(* CODESYS project 3v12manLoadTestPLC.project

Project tree, tasks and I/O mapping:
  Device : Owen SPK2xx 03.CS.WEB, Owen, order no. 023, version 3.5.4.20
    application Application
      task MainTask (cyclic, interval t#20ms, priority 1) calls PLC_PRG
      task VISU_TASK (cyclic, interval 100 ms, priority 31) calls VisuElems.Visu_Prg
      program PLC_PRG [ST]: actNextUnloadStep, actInit, outWriteVars, autoLoadHopper, autoUnloadHopper, actTimeCounting, sysAutoStat, sysManStat, manLoad, manUnload, inReadVars, setTara, actLoadSwitches, actUnloadSwitches, pause, chkEngines
      image pool ImagePool
      data type TableStruct
      Functions/
        function TimeInput [ST]
        function two_word_to_real [ST]
        function block NoiseFilter [ST]: isInEdges, setEdges, setAccuracy, refresh
      GlobalVarList/
        global variables GVL
        global variables ArrayList
        global variables TimeVars
        global variables CurrentValues
      Windows/
        visualisation Visualization
        visualisation ManualInput
        visualisation Settings
        visualisation AutoWork
        visualisation LoadProcessWindow
        visualisation LoadingFinished
        visualisation UnloadProcessWindow
        visualisation RepeatOrNewPRG
        visualisation TimeCounter
        Dialogs/
          visualisation DialogLoad
          visualisation Alarm
        visualisation TmpUnused
        visualisation SystemSettings
      Managers/
        libraries: VisuDialogs, * (System); CmpSysExec, 1.0.0.2 (Owen); SPK_Tools, 1.0.1 (Owen); RS mode library, 1.0.0.0 (Owen); ArchiverSPK, 3.5.3.53 (Owen); CAA File, 3.5.5.0 (CAA Technical Workgroup); Time and Date, 3.5.1.0 (3S - Smart Software Solutions GmbH); Standard, * (System); Mx110Assistant, 3.5.4.0 (Owen)
        RecipeManager
          recipe definition Receipt: arrayOfIngr[0].stepNum : STRING; arrayOfIngr[0].nameOfIngr : STRING; arrayOfIngr[0].weightOfIngr : STRING; arrayOfIngr[0].isDissolve : STRING; arrayOfIngr[0].timeOfMixing : STRING; arrayOfIngr[0].addMessage : STRING; arrayOfIngr[1].stepNum : STRING; arrayOfIngr[1].nameOfIngr : STRING; arrayOfIngr[1].weightOfIngr : STRING; arrayOfIngr[1].isDissolve : STRING; arrayOfIngr[1].timeOfMixing : STRING; arrayOfIngr[1].addMessage : STRING; arrayOfIngr[2].stepNum : STRING; arrayOfIngr[2].nameOfIngr : STRING; arrayOfIngr[2].weightOfIngr : STRING; arrayOfIngr[2].isDissolve : STRING; arrayOfIngr[2].timeOfMixing : STRING; arrayOfIngr[2].addMessage : STRING; arrayOfIngr[3].stepNum : STRING; arrayOfIngr[3].nameOfIngr : STRING; arrayOfIngr[3].weightOfIngr : STRING; arrayOfIngr[3].isDissolve : STRING; arrayOfIngr[3].timeOfMixing : STRING; arrayOfIngr[3].addMessage : STRING; arrayOfIngr[4].stepNum : STRING; arrayOfIngr[4].nameOfIngr : STRING; arrayOfIngr[4].weightOfIngr : STRING; arrayOfIngr[4].isDissolve : STRING; arrayOfIngr[4].timeOfMixing : STRING; arrayOfIngr[4].addMessage : STRING; arrayOfIngr[5].stepNum : STRING; arrayOfIngr[5].nameOfIngr : STRING; arrayOfIngr[5].weightOfIngr : STRING; arrayOfIngr[5].isDissolve : STRING; arrayOfIngr[5].timeOfMixing : STRING; arrayOfIngr[5].addMessage : STRING; arrayOfIngr[6].stepNum : STRING; arrayOfIngr[6].nameOfIngr : STRING; arrayOfIngr[6].weightOfIngr : STRING; arrayOfIngr[6].isDissolve : STRING; arrayOfIngr[6].timeOfMixing : STRING; arrayOfIngr[6].addMessage : STRING; arrayOfIngr[7].stepNum : STRING; arrayOfIngr[7].nameOfIngr : STRING; arrayOfIngr[7].weightOfIngr : STRING; arrayOfIngr[7].isDissolve : STRING; arrayOfIngr[7].timeOfMixing : STRING; arrayOfIngr[7].addMessage : STRING; arrayOfIngr[8].stepNum : STRING; arrayOfIngr[8].nameOfIngr : STRING; arrayOfIngr[8].weightOfIngr : STRING; arrayOfIngr[8].isDissolve : STRING; arrayOfIngr[8].timeOfMixing : STRING; arrayOfIngr[8].addMessage : STRING; arrayOfIngr[9].stepNum : STRING; arrayOfIngr[9].nameOfIngr : STRING; arrayOfIngr[9].weightOfIngr : STRING; arrayOfIngr[9].isDissolve : STRING; arrayOfIngr[9].timeOfMixing : STRING; arrayOfIngr[9].addMessage : STRING; arrayOfIngr[10].stepNum : STRING; arrayOfIngr[10].nameOfIngr : STRING; arrayOfIngr[10].weightOfIngr : STRING; arrayOfIngr[10].isDissolve : STRING; arrayOfIngr[10].timeOfMixing : STRING; arrayOfIngr[10].addMessage : STRING; arrayOfIngr[11].stepNum : STRING; arrayOfIngr[11].nameOfIngr : STRING; arrayOfIngr[11].weightOfIngr : STRING; arrayOfIngr[11].isDissolve : STRING; arrayOfIngr[11].timeOfMixing : STRING; arrayOfIngr[11].addMessage : STRING; arrayOfIngr[12].stepNum : STRING; arrayOfIngr[12].nameOfIngr : STRING; arrayOfIngr[12].weightOfIngr : STRING; arrayOfIngr[12].isDissolve : STRING; arrayOfIngr[12].timeOfMixing : STRING; arrayOfIngr[12].addMessage : STRING; arrayOfIngr[13].stepNum : STRING; arrayOfIngr[13].nameOfIngr : STRING; arrayOfIngr[13].weightOfIngr : STRING; arrayOfIngr[13].isDissolve : STRING; arrayOfIngr[13].timeOfMixing : STRING; arrayOfIngr[13].addMessage : STRING; arrayOfIngr[14].stepNum : STRING; arrayOfIngr[14].nameOfIngr : STRING; arrayOfIngr[14].weightOfIngr : STRING; arrayOfIngr[14].isDissolve : STRING; arrayOfIngr[14].timeOfMixing : STRING; arrayOfIngr[14].addMessage : STRING; arrayOfIngr[15].stepNum : STRING; arrayOfIngr[15].nameOfIngr : STRING; arrayOfIngr[15].weightOfIngr : STRING; arrayOfIngr[15].isDissolve : STRING; arrayOfIngr[15].timeOfMixing : STRING; arrayOfIngr[15].addMessage : STRING; arrayOfIngr[16].stepNum : STRING; arrayOfIngr[16].nameOfIngr : STRING; arrayOfIngr[16].weightOfIngr : STRING; arrayOfIngr[16].isDissolve : STRING; arrayOfIngr[16].timeOfMixing : STRING; arrayOfIngr[16].addMessage : STRING; arrayOfIngr[17].stepNum : STRING; arrayOfIngr[17].nameOfIngr : STRING; arrayOfIngr[17].weightOfIngr : STRING; arrayOfIngr[17].isDissolve : STRING; arrayOfIngr[17].timeOfMixing : STRING; arrayOfIngr[17].addMessage : STRING; arrayOfIngr[18].stepNum : STRING; arrayOfIngr[18].nameOfIngr : STRING; arrayOfIngr[18].weightOfIngr : STRING; arrayOfIngr[18].isDissolve : STRING; arrayOfIngr[18].timeOfMixing : STRING; arrayOfIngr[18].addMessage : STRING; arrayOfIngr[19].stepNum : STRING; arrayOfIngr[19].nameOfIngr : STRING; arrayOfIngr[19].weightOfIngr : STRING; arrayOfIngr[19].isDissolve : STRING; arrayOfIngr[19].timeOfMixing : STRING; arrayOfIngr[19].addMessage : STRING; arrayOfIngr[20].stepNum : STRING; arrayOfIngr[20].nameOfIngr : STRING; arrayOfIngr[20].weightOfIngr : STRING; arrayOfIngr[20].isDissolve : STRING; arrayOfIngr[20].timeOfMixing : STRING; arrayOfIngr[20].addMessage : STRING; arrayOfIngr[21].stepNum : STRING; arrayOfIngr[21].nameOfIngr : STRING; arrayOfIngr[21].weightOfIngr : STRING; arrayOfIngr[21].isDissolve : STRING; arrayOfIngr[21].timeOfMixing : STRING; arrayOfIngr[21].addMessage : STRING; arrayOfIngr[22].stepNum : STRING; arrayOfIngr[22].nameOfIngr : STRING; arrayOfIngr[22].weightOfIngr : STRING; arrayOfIngr[22].isDissolve : STRING; arrayOfIngr[22].timeOfMixing : STRING; arrayOfIngr[22].addMessage : STRING; arrayOfIngr[23].stepNum : STRING; arrayOfIngr[23].nameOfIngr : STRING; arrayOfIngr[23].weightOfIngr : STRING; arrayOfIngr[23].isDissolve : STRING; arrayOfIngr[23].timeOfMixing : STRING; arrayOfIngr[23].addMessage : STRING; arrayOfIngr[24].stepNum : STRING; arrayOfIngr[24].nameOfIngr : STRING; arrayOfIngr[24].weightOfIngr : STRING; arrayOfIngr[24].isDissolve : STRING; arrayOfIngr[24].timeOfMixing : STRING; arrayOfIngr[24].addMessage : STRING; arrayOfIngr[25].stepNum : STRING; arrayOfIngr[25].nameOfIngr : STRING; arrayOfIngr[25].weightOfIngr : STRING; arrayOfIngr[25].isDissolve : STRING; arrayOfIngr[25].timeOfMixing : STRING; arrayOfIngr[25].addMessage : STRING; arrayOfIngr[26].stepNum : STRING; arrayOfIngr[26].nameOfIngr : STRING; arrayOfIngr[26].weightOfIngr : STRING; arrayOfIngr[26].isDissolve : STRING; arrayOfIngr[26].timeOfMixing : STRING; arrayOfIngr[26].addMessage : STRING; arrayOfIngr[27].stepNum : STRING; arrayOfIngr[27].nameOfIngr : STRING; arrayOfIngr[27].weightOfIngr : STRING; arrayOfIngr[27].isDissolve : STRING; arrayOfIngr[27].timeOfMixing : STRING; arrayOfIngr[27].addMessage : STRING; arrayOfIngr[28].stepNum : STRING; arrayOfIngr[28].nameOfIngr : STRING; arrayOfIngr[28].weightOfIngr : STRING; arrayOfIngr[28].isDissolve : STRING; arrayOfIngr[28].timeOfMixing : STRING; arrayOfIngr[28].addMessage : STRING; arrayOfIngr[29].stepNum : STRING; arrayOfIngr[29].nameOfIngr : STRING; arrayOfIngr[29].weightOfIngr : STRING; arrayOfIngr[29].isDissolve : STRING; arrayOfIngr[29].timeOfMixing : STRING; arrayOfIngr[29].addMessage : STRING; arrayOfIngr[30].stepNum : STRING; arrayOfIngr[30].nameOfIngr : STRING; arrayOfIngr[30].weightOfIngr : STRING; arrayOfIngr[30].isDissolve : STRING; arrayOfIngr[30].timeOfMixing : STRING; arrayOfIngr[30].addMessage : STRING; arrayOfIngr[31].stepNum : STRING; arrayOfIngr[31].nameOfIngr : STRING; arrayOfIngr[31].weightOfIngr : STRING; arrayOfIngr[31].isDissolve : STRING; arrayOfIngr[31].timeOfMixing : STRING; arrayOfIngr[31].addMessage : STRING; arrayOfIngr[32].stepNum : STRING; arrayOfIngr[32].nameOfIngr : STRING; arrayOfIngr[32].weightOfIngr : STRING; arrayOfIngr[32].isDissolve : STRING; arrayOfIngr[32].timeOfMixing : STRING; arrayOfIngr[32].addMessage : STRING; arrayOfIngr[33].stepNum : STRING; arrayOfIngr[33].nameOfIngr : STRING; arrayOfIngr[33].weightOfIngr : STRING; arrayOfIngr[33].isDissolve : STRING; arrayOfIngr[33].timeOfMixing : STRING; arrayOfIngr[33].addMessage : STRING; arrayOfIngr[34].stepNum : STRING; arrayOfIngr[34].nameOfIngr : STRING; arrayOfIngr[34].weightOfIngr : STRING; arrayOfIngr[34].isDissolve : STRING; arrayOfIngr[34].timeOfMixing : STRING; arrayOfIngr[34].addMessage : STRING; arrayOfIngr[35].stepNum : STRING; arrayOfIngr[35].nameOfIngr : STRING; arrayOfIngr[35].weightOfIngr : STRING; arrayOfIngr[35].isDissolve : STRING; arrayOfIngr[35].timeOfMixing : STRING; arrayOfIngr[35].addMessage : STRING; arrayOfIngr[36].stepNum : STRING; arrayOfIngr[36].nameOfIngr : STRING; arrayOfIngr[36].weightOfIngr : STRING; arrayOfIngr[36].isDissolve : STRING; arrayOfIngr[36].timeOfMixing : STRING; arrayOfIngr[36].addMessage : STRING; arrayOfIngr[37].stepNum : STRING; arrayOfIngr[37].nameOfIngr : STRING; arrayOfIngr[37].weightOfIngr : STRING; arrayOfIngr[37].isDissolve : STRING; arrayOfIngr[37].timeOfMixing : STRING; arrayOfIngr[37].addMessage : STRING; arrayOfIngr[38].stepNum : STRING; arrayOfIngr[38].nameOfIngr : STRING; arrayOfIngr[38].weightOfIngr : STRING; arrayOfIngr[38].isDissolve : STRING; arrayOfIngr[38].timeOfMixing : STRING; arrayOfIngr[38].addMessage : STRING; arrayOfIngr[39].stepNum : STRING; arrayOfIngr[39].nameOfIngr : STRING; arrayOfIngr[39].weightOfIngr : STRING; arrayOfIngr[39].isDissolve : STRING; arrayOfIngr[39].timeOfMixing : STRING; arrayOfIngr[39].addMessage : STRING; arrayOfIngr[40].stepNum : STRING; arrayOfIngr[40].nameOfIngr : STRING; arrayOfIngr[40].weightOfIngr : STRING; arrayOfIngr[40].isDissolve : STRING; arrayOfIngr[40].timeOfMixing : STRING; arrayOfIngr[40].addMessage : STRING; arrayOfIngr[41].stepNum : STRING; arrayOfIngr[41].nameOfIngr : STRING; arrayOfIngr[41].weightOfIngr : STRING; arrayOfIngr[41].isDissolve : STRING; arrayOfIngr[41].timeOfMixing : STRING; arrayOfIngr[41].addMessage : STRING; arrayOfIngr[42].stepNum : STRING; arrayOfIngr[42].nameOfIngr : STRING; arrayOfIngr[42].weightOfIngr : STRING; arrayOfIngr[42].isDissolve : STRING; arrayOfIngr[42].timeOfMixing : STRING; arrayOfIngr[42].addMessage : STRING; arrayOfIngr[43].stepNum : STRING; arrayOfIngr[43].nameOfIngr : STRING; arrayOfIngr[43].weightOfIngr : STRING; arrayOfIngr[43].isDissolve : STRING; arrayOfIngr[43].timeOfMixing : STRING; arrayOfIngr[43].addMessage : STRING; arrayOfIngr[44].stepNum : STRING; arrayOfIngr[44].nameOfIngr : STRING; arrayOfIngr[44].weightOfIngr : STRING; arrayOfIngr[44].isDissolve : STRING; arrayOfIngr[44].timeOfMixing : STRING; arrayOfIngr[44].addMessage : STRING; arrayOfIngr[45].stepNum : STRING; arrayOfIngr[45].nameOfIngr : STRING; arrayOfIngr[45].weightOfIngr : STRING; arrayOfIngr[45].isDissolve : STRING; arrayOfIngr[45].timeOfMixing : STRING; arrayOfIngr[45].addMessage : STRING; arrayOfIngr[46].stepNum : STRING; arrayOfIngr[46].nameOfIngr : STRING; arrayOfIngr[46].weightOfIngr : STRING; arrayOfIngr[46].isDissolve : STRING; arrayOfIngr[46].timeOfMixing : STRING; arrayOfIngr[46].addMessage : STRING; arrayOfIngr[47].stepNum : STRING; arrayOfIngr[47].nameOfIngr : STRING; arrayOfIngr[47].weightOfIngr : STRING; arrayOfIngr[47].isDissolve : STRING; arrayOfIngr[47].timeOfMixing : STRING; arrayOfIngr[47].addMessage : STRING; arrayOfIngr[48].stepNum : STRING; arrayOfIngr[48].nameOfIngr : STRING; arrayOfIngr[48].weightOfIngr : STRING; arrayOfIngr[48].isDissolve : STRING; arrayOfIngr[48].timeOfMixing : STRING; arrayOfIngr[48].addMessage : STRING; arrayOfIngr[49].stepNum : STRING; arrayOfIngr[49].nameOfIngr : STRING; arrayOfIngr[49].weightOfIngr : STRING; arrayOfIngr[49].isDissolve : STRING; arrayOfIngr[49].timeOfMixing : STRING; arrayOfIngr[49].addMessage : STRING; arrayOfIngr[50].stepNum : STRING; arrayOfIngr[50].nameOfIngr : STRING; arrayOfIngr[50].weightOfIngr : STRING; arrayOfIngr[50].isDissolve : STRING; arrayOfIngr[50].timeOfMixing : STRING; arrayOfIngr[50].addMessage : STRING
      Classes/
        function block List [ST]: getPrgIdx, getLineFromPrgArr, checkPrgArr, clearList, clearLine, writeLine
        function block DiscrSwitch [ST]: allOff, set, setLaterOn, setLaterOff, unloadOn, unloadLaterOff, unloadOff
        function block Checker [ST]: isHopperEmpty, isPrgActive
        function block Way [ST]: getWay, tmpLimitWay, getWayId, setWay, setIdx
    COM_2 : Modbus COM, 3S - Smart Software Solutions GmbH, version 3.4.0.0
        settings: DataBits = 8; StopBits = 1; ComPort = 3
      Modbus_Master_COM_Port_2 : Modbus Master, COM Port, 3S - Smart Software Solutions GmbH, version 3.5.5.0
          settings: Transmission = 'RTU'; ResponseTimeout = 300; TimeBetweenFrames = 20; Auto-restart communication = TRUE
        Out_MU110_16R : Modbus Slave, COM Port, 3S - Smart Software Solutions GmbH, version 3.5.4.0
            settings: SlaveAddress = 17; ResponseTimeout = 300; UseExtendedFunctionCodes = TRUE; Channel 0.Function Code = 16; Channel 0.Read Offset = 0; Channel 0.Read Length = 0; Channel 0.Write Offset = 16#0032; Channel 0.Write Length = 1; Channel 0.Cycle Time = 100
            output Application.iOutDiscrets : ARRAY[0..0] OF WORD  // Channel 0
        In_MV110_16D : Modbus Slave, COM Port, 3S - Smart Software Solutions GmbH, version 3.5.4.0
            settings: SlaveAddress = 1; ResponseTimeout = 300; UseExtendedFunctionCodes = TRUE; Channel 0.Function Code = 3; Channel 0.Read Offset = 16#0033; Channel 0.Read Length = 1; Channel 0.Write Offset = 0; Channel 0.Write Length = 0; Channel 0.Cycle Time = 100
            input  Application.iInDiscrets : ARRAY[0..0] OF WORD  // Channel 0
    COM_3 : Modbus COM, 3S - Smart Software Solutions GmbH, version 3.4.0.0
        settings: DataBits = 8; StopBits = 1; ComPort = 4
      Modbus_Master_COM_Port : Modbus Master, COM Port, 3S - Smart Software Solutions GmbH, version 3.5.5.0
          settings: Transmission = 'RTU'; ResponseTimeout = 300; TimeBetweenFrames = 10; Auto-restart communication = TRUE
        MV110_1TD : MV110-1TD, Owen, order no. 3.5.4.1, version 3.5.4.0
            settings: SlaveAddress = 1; ResponseTimeout = 300; UseExtendedFunctionCodes = TRUE
            unmapped channels: Rd.fF1, Rd.St, in1, out1
  text list GlobalTextList
  GlobalImagePool
  image pool ImagePool
  5ce3da45-db07-42e7-a21c-a00fff4ed8f6|C:\Users\Валентин\Desktop\home.png
  5ce3da45-db07-42e7-a21c-a00fff4ed8f6|D:\Pictures\tanzania.jpg
  5ce3da45-db07-42e7-a21c-a00fff4ed8f6|D:\Pictures\tanzania800x480.jpg
  5ce3da45-db07-42e7-a21c-a00fff4ed8f6|D:\Pictures\BeachHouse800x480.jpg
  5ce3da45-db07-42e7-a21c-a00fff4ed8f6|D:\Projects\OWEN\JAVA\GIT\settings.png
  5ce3da45-db07-42e7-a21c-a00fff4ed8f6|D:\Projects\OWEN\PIC\motherboard.png
  5ce3da45-db07-42e7-a21c-a00fff4ed8f6|D:\Projects\OWEN\PIC\home.png
  5ce3da45-db07-42e7-a21c-a00fff4ed8f6|D:\Projects\OWEN\PIC\settings.jpg
  5ce3da45-db07-42e7-a21c-a00fff4ed8f6|D:\Projects\OWEN\PIC\reset.jpg
  5ce3da45-db07-42e7-a21c-a00fff4ed8f6|D:\Projects\OWEN\PIC\reset.png
  5ce3da45-db07-42e7-a21c-a00fff4ed8f6|D:\Projects\OWEN\PIC\resetButton.png
  5ce3da45-db07-42e7-a21c-a00fff4ed8f6|D:\Projects\OWEN\PIC\start.png
  5ce3da45-db07-42e7-a21c-a00fff4ed8f6|D:\Projects\OWEN\PIC\remove.png
  5ce3da45-db07-42e7-a21c-a00fff4ed8f6|D:\Projects\OWEN\PIC\ok.png
  5ce3da45-db07-42e7-a21c-a00fff4ed8f6|D:\Projects\OWEN\PIC\cancel.png
  function block Time_Struct [ST]
  5ce3da45-db07-42e7-a21c-a00fff4ed8f6|D:\Projects\OWEN\PIC\add.png
  5ce3da45-db07-42e7-a21c-a00fff4ed8f6|D:\Projects\OWEN\PIC\back.png
  5ce3da45-db07-42e7-a21c-a00fff4ed8f6|D:\Projects\OWEN\PIC\next.png
  5ce3da45-db07-42e7-a21c-a00fff4ed8f6|D:\Projects\OWEN\PIC\Drives-Downloads-icon.png
  5ce3da45-db07-42e7-a21c-a00fff4ed8f6|D:\Projects\OWEN\PIC\Actions-application-exit-icon.png
  5ce3da45-db07-42e7-a21c-a00fff4ed8f6|D:\Projects\OWEN\PIC\App-desktop-enhancements-icon.png
  5ce3da45-db07-42e7-a21c-a00fff4ed8f6|D:\Projects\OWEN\PIC\chemistryS.png
  5ce3da45-db07-42e7-a21c-a00fff4ed8f6|D:\Projects\OWEN\PIC\chemistry.png
  5ce3da45-db07-42e7-a21c-a00fff4ed8f6|D:\Projects\OWEN\PIC\Iconshock-Real-Vista-Education-Laboratory.png
  5ce3da45-db07-42e7-a21c-a00fff4ed8f6|D:\Projects\OWEN\PIC\pause.png
  5ce3da45-db07-42e7-a21c-a00fff4ed8f6|D:\Projects\OWEN\PIC\startAgain.png
  5ce3da45-db07-42e7-a21c-a00fff4ed8f6|D:\Projects\OWEN\PIC\start-button-305427_960_720.png
  5ce3da45-db07-42e7-a21c-a00fff4ed8f6|D:\Projects\OWEN\PIC\repeat.png
  5ce3da45-db07-42e7-a21c-a00fff4ed8f6|D:\Projects\OWEN\PIC\download.png
  5ce3da45-db07-42e7-a21c-a00fff4ed8f6|D:\Projects\OWEN\PIC\upload.png
*)

// Device/Application/TableStruct
TYPE TableStruct :
STRUCT
	stepNum:STRING;
	nameOfIngr:STRING;
	weightOfIngr:STRING;
	isDissolve:STRING;
	timeOfMixing:STRING;
	addMessage:STRING;	
END_STRUCT
END_TYPE

// Device/Application/GlobalVarList/GVL
VAR_GLOBAL
	iOutDiscrets: INT;
	iInDiscrets:INT;
	ON : BOOL := TRUE;
	OFF : BOOL := FALSE;	
	arr1:ARRAY[0..1]OF WORD;		
	arr2:ARRAY[0..1]OF WORD;
	arr3:ARRAY[0..1]OF WORD;
	arr4:ARRAY[0..1]OF WORD;	
END_VAR

// Device/Application/GlobalVarList/ArrayList
VAR_GLOBAL
	ListOfPrgNames: ARRAY[0..100] OF STRING;	
	ptToListPrg: POINTER TO ARRAY [0..100] OF STRING := ADR(ListOfPrgNames);
	arrayOfIngr: ARRAY[0..50] OF TableStruct;
	tempArrOfIngr: ARRAY[0..100] OF TableStruct;		
END_VAR

// Device/Application/GlobalVarList/TimeVars
VAR_GLOBAL
	timerActive:BOOL := FALSE;
	strTimer:STRING;
	inputTime:DWORD;
END_VAR

// Device/Application/GlobalVarList/CurrentValues
VAR_GLOBAL
	currentPrgSteps:INT;	
	currentProgramIdx:INT;
	currentPrgName: STRING;
	currentIngredientName: STRING;
	currentWeight: INT;
	currentPoint : INT;
//	strCrntWay: STRING;
	message: STRING;	
	currentTimeMixing: TIME;
END_VAR

// Device/Application/PLC_PRG
PROGRAM PLC_PRG
VAR
	iMaxWeight: INT := 1000;	

	tOn1:TON;
	tOn2:TON;
	tCheckDelay:TON;
	
	switch:DiscrSwitch;
	ptSwitch: POINTER TO DiscrSwitch := ADR(switch);
	timeStruct:Time_Struct;	
	bTimerActive:BOOL := FALSE;
	strTimer:STRING;
	dwInTime:DWORD;
	rWeight:REAL;
	
	list:List;
	checker:Checker;
	signalFilter:NoiseFilter;

	strResipesExt:STRING := 'Receipt';
	RecManager:RecipeManCommands;

	bInit:BOOL := TRUE;
	bPause:BOOL;
	bRunOnce:BOOL;
	bLoadDone:BOOL;
	bManLoadDone:BOOL;
	bMsgVisible:BOOL := TRUE;
	bManMode: BOOL;
	
	iTotalIngrWeight:INT;
	iErrEngineNum:INT := 0;
	
	x: INT := 0;
	iEdge: INT := 1000;
	bSwitch: BOOL;
	bLamp: BOOL;	

	data0:REAL;
END_VAR
VAR RETAIN
	rTara:REAL;	
END_VAR

inReadVars();

IF bInit THEN // run once
	actInit();END_IF


IF bManMode THEN
	sysManStat();
ELSE
	sysAutoStat();
END_IF
outWriteVars();

chkEngines();
//data0:=two_word_to_real(ADR(arr1));

ACTION actNextUnloadStep:
bTimerActive := FALSE;
VisuElems.CURRENTVISU := 'UnloadProcessWindow';
currentProgramIdx := currentProgramIdx + 1;
list.getLineFromPrgArr(currentProgramIdx);
IF currentPrgSteps >= currentProgramIdx THEN
		 VisuElems.CURRENTVISU := 'RepeatOrNewPRG';
		 bLoadDone := FALSE;
END_IF
END_ACTION

ACTION actInit:
RecManager.ReloadRecipes(strResipesExt);
RecManager.GetRecipeNames(strResipesExt, ptToListPrg, 100,0);
list(ptToSwitch := ptSwitch);
bInit := FALSE;
END_ACTION

ACTION outWriteVars:

iOutDiscrets := Switch.iOut;
END_ACTION

ACTION autoLoadHopper:
IF bSwitch THEN
  IF x < currentPoint + currentWeight AND x < iMaxWeight THEN 
	 bMsgVisible := FALSE;
	 switch.set(ON);
	 pause();
//	 x := x + 1;	 
  ELSE 
	switch.set(OFF);
	actLoadSwitches();
	IF tOn2.Q THEN
 		currentPoint := currentPoint + currentWeight;
 		IF x >= currentPoint AND currentPrgSteps - 1 > currentProgramIdx THEN
	 		currentProgramIdx := currentProgramIdx + 1;
	 		list.getLineFromPrgArr(currentProgramIdx);
		 ELSIF currentPrgSteps >= currentProgramIdx THEN
		 	currentProgramIdx := 0;
		 	list.getLineFromPrgArr(currentProgramIdx);
		 	bLoadDone:=TRUE;
		 	VisuElems.CURRENTVISU := 'LoadingFinished';
		END_IF
 		bMsgVisible := TRUE;
		bSwitch := FALSE;		
	END_IF
 END_IF
END_IF
END_ACTION

ACTION autoUnloadHopper:
IF bSwitch THEN
  IF x > currentPoint - currentWeight AND x > 0 THEN 
	 bMsgVisible := FALSE;
//	 x := x - 1;
	 Switch.unloadOn();
  ELSE
	actUnloadSwitches();
	IF tOn1.Q THEN	 
 	currentPoint:= currentPoint - currentWeight;
 		IF x >= currentPoint AND currentPrgSteps - 1 >= currentProgramIdx THEN
			VisuElems.CURRENTVISU := 'TimeCounter';
			bTimerActive:=TRUE;	  
		END_IF
 	bMsgVisible := TRUE;
 	bSwitch:= FALSE;
	tOn1(IN := FALSE);
	END_IF	
 END_IF
END_IF
END_ACTION

ACTION actTimeCounting:
IF TIME_TO_REAL(currentTimeMixing) >= 0 THEN
 	currentTimeMixing := REAL_TO_TIME ( TIME_TO_REAL(currentTimeMixing) - 20); 
	timeStruct(Type_Time := currentTimeMixing);
	strTimer:=CONCAT(CONCAT(DWORD_TO_STRING(timeStruct.Minute),'m:'),CONCAT(DWORD_TO_STRING(timeStruct.Second),'s'));
		IF TIME_TO_REAL(currentTimeMixing) = 0 THEN
			actNextUnloadStep();
		END_IF	
END_IF
END_ACTION

ACTION sysAutoStat:
IF bTimerActive THEN 
	actTimeCounting(); 
END_IF

IF bLoadDone THEN	
	autoUnloadHopper();
ELSE	
	autoLoadHopper();
END_IF
END_ACTION

ACTION sysManStat:
IF bManLoadDone THEN	
	manUnload();
ELSE
	manLoad();
END_IF
END_ACTION

ACTION manLoad:
IF bRunOnce THEN
		tOn1(IN := FALSE);
		list.way.getWay();
		switch(iWayIdx := list.way.getWayId());
		bRunOnce := FALSE;
END_IF
IF bSwitch THEN	
  IF x < currentWeight AND x < iMaxWeight THEN 
	Switch.set(ON);	
//	x := x + 1;	 
  ELSE
	switch.set(OFF);
//actLoadSwitches();
 END_IF
END_IF
END_ACTION

ACTION manUnload:
IF bSwitch THEN
  IF x > 0 THEN 
	 switch.unloadOn();
//	 x := x - 1;	 
  ELSE
	  
	//switch.unloadOff();
	actUnloadSwitches();
	tOn1(IN := bSwitch);
 END_IF
END_IF
END_ACTION

ACTION inReadVars:
rWeight := MV110_1TD.RdfF1 - rTara;
signalFilter(rIn := rWeight, rOut => rWeight);
x := REAL_TO_INT(rWeight);
//IF iInDiscrets.0 THEN
	//bSwitch := TRUE;
//END_IF
switch(iIn := iInDiscrets);
END_ACTION

ACTION setTara:
rTara := MV110_1TD.RdfF1;
signalFilter.refresh();
END_ACTION

ACTION actLoadSwitches:
switch.set(OFF);
tOn1(IN := TRUE, PT := T#1S);
switch.setLaterOn(tOn1.Q);
tOn2(IN := tOn1.Q, PT := T#10S);
	IF tOn2.Q THEN
		switch.setLaterOff(OFF);
		bSwitch := FALSE;
		tOn1(IN := FALSE);
	END_IF
END_ACTION

ACTION actUnloadSwitches:
switch.set(OFF);
switch.unloadOff();
tOn1(IN := TRUE, PT := T#10S);	  	  
 	IF tOn1.Q THEN
	 Switch.unloadLaterOff(OFF);
	 bSwitch := FALSE;
	END_IF
END_ACTION

ACTION pause:
IF bPause THEN
	switch.allOff();
END_IF
END_ACTION

ACTION chkEngines:
// проверка подключения автоматов защиты двигателей
tCheckDelay(PT := T#10s, IN := TRUE);
IF tCheckDelay.Q THEN
	IF NOT switch.iIn.12 THEN
		switch.allOff();
		iErrEngineNum := 13;
		VisuElems.CURRENTVISU := 'Alarm';	
	END_IF
	IF NOT switch.iIn.13 THEN	
		switch.allOff();
		iErrEngineNum := 14;
		VisuElems.CURRENTVISU := 'Alarm';	
	END_IF
	IF NOT switch.iIn.14 THEN	
		switch.allOff();
		iErrEngineNum := 15;
		VisuElems.CURRENTVISU := 'Alarm';	
	END_IF
	IF NOT switch.iIn.15 THEN	
		switch.allOff();
		iErrEngineNum := 16;
		VisuElems.CURRENTVISU := 'Alarm';	
	END_IF
END_IF
END_ACTION

END_PROGRAM

// Device/Application/Functions/two_word_to_real
FUNCTION two_word_to_real : REAL
VAR_INPUT
	in_data: POINTER TO ARRAY[0..1]OF WORD;
END_VAR
VAR
	p1:POINTER TO BYTE;
	p2:POINTER TO BYTE;
END_VAR

p1:=ADR(two_word_to_real);
p2:=ADR(in_data^[1]);

p1^:=p2^;
p1:=p1+1;
p2:=p2+1;
p1^:=p2^;
p1:=p1+1;
p2:=ADR(in_data^[0]);
p1^:=p2^;
p1:=p1+1;
p2:=p2+1;
p1^:=p2^;

END_FUNCTION

// Device/Application/Classes/DiscrSwitch

FUNCTION_BLOCK PUBLIC DiscrSwitch
VAR_INPUT
	iIn:INT;	
	iWayIdx:INT;
END_VAR
VAR_OUTPUT
	iOut:INT;
END_VAR

//выключает все 16 переключателей
METHOD allOff
VAR_INPUT
END_VAR
iOut := 0;
END_METHOD

//устанавливает выключатели в ON немедленно
METHOD PUBLIC set
VAR_INPUT
	bInput:BOOL;
END_VAR
CASE iWayIdx OF //набор переключателей в зависимости от текущего пути
	0:// путь по умолчанию		
			iOut.12 := bInput; // двигатель
			iOut.0 := bInput;  //задвижка
			
	1:// путь через вибросито
			iOut.0 := bInput; // двигатель
			iOut.1 := bInput; // двигатель
			iOut.9 := bInput;  //задвижка
			
	2..10://через BigBag
	;
	
END_CASE
END_METHOD

//устанавливает выключатели в ON через интервал
METHOD PUBLIC setLaterOn
VAR_INPUT
	bInput:BOOL;
END_VAR
VAR
END_VAR
CASE iWayIdx OF //набор переключателей в зависимости от текущего пути
	0:// путь по умолчанию
			iOut.3 := bInput; // двигатель					
			iOut.7 := bInput; //распределитель
			iOut.11 := bInput;  //задвижка	
	1:// путь через вибросито
//			iOut.0 := bInput;//двигатель	
			iOut.1 := bInput;  //двигатель
			iOut.6 := bInput; //распределитель
			iOut.9 := bInput;  //задвижка	
	2..10:
	;
	
	ELSE
		;//выброс ошибки на недопустимый параметр	
END_CASE
END_METHOD

//устанавливает выключатели в OFF через интервал
METHOD PUBLIC setLaterOff
VAR_INPUT
	bInput:BOOL;
END_VAR
CASE iWayIdx OF //набор переключателей в зависимости от текущего пути
	0:// путь по умолчанию
			iOut.3 := bInput; // двигатель					
			iOut.7 := bInput; //распределитель
			iOut.11 := bInput;  //задвижка	
	1:// путь через вибросито
//			iOut.0 := bInput;//двигатель	
			iOut.1 := bInput;  //двигатель
			iOut.6 := bInput; //распределитель
			iOut.9 := bInput;  //задвижка
	2..10:
	;
	
	ELSE
		;//выброс ошибки на недопустимый параметр	
END_CASE
END_METHOD

METHOD PUBLIC unloadOn
VAR_INPUT
END_VAR
iOut.1 := TRUE;
iOut.15 := TRUE;
END_METHOD

METHOD unloadLaterOff
VAR_INPUT
	bInput:BOOL;
END_VAR
iOut.15 := bInput;
END_METHOD

METHOD PUBLIC unloadOff
VAR_INPUT
END_VAR
iOut.1 := FALSE;
END_METHOD

END_FUNCTION_BLOCK

// Time_Struct
FUNCTION_BLOCK Time_Struct
VAR_INPUT
	Type_Time:TIME;
END_VAR
VAR_OUTPUT
	Day:DWORD;
	Hour:DWORD;
	Minute:DWORD;
	Second:DWORD;
	Millisecond:DWORD;  
END_VAR
VAR
		Time_DWORD:DWORD;
		Day_Ost:DWORD;
		Hour_Ost:DWORD;
		Minute_Ost:DWORD;
		Second_Ost:DWORD;
		Millisecond_Ost:DWORD; 
END_VAR


Time_DWORD := TIME_TO_DWORD(Type_Time);

Millisecond := Second_Ost;

Second := Minute_Ost/ 1000;
Second_Ost := Minute_Ost MOD 1000;

Minute := Hour_Ost/60000;
Minute_Ost := Hour_Ost MOD 60000;

Hour := Day_Ost/3600000;
Hour_Ost := Day_Ost MOD 3600000;

Day := Time_DWORD/86400000;
Day_Ost := Time_DWORD MOD 86400000;

END_FUNCTION_BLOCK

// Device/Application/Classes/List
FUNCTION_BLOCK List
VAR_INPUT
	ptToSwitch:POINTER TO DiscrSwitch;		
END_VAR
VAR_OUTPUT
END_VAR
VAR	
	way:Way;
	iLinePrgList:INT;
	iLine:INT;	
	iArrLength: INT := 50;
	iPrgAmount:INT := 100;	
	iTotalWeight:INT;
	iCleanIdx:INT;
END_VAR

METHOD getPrgIdx : INT
VAR_INPUT
END_VAR
getPrgIdx := iLinePrgList;
END_METHOD

METHOD PUBLIC getLineFromPrgArr : BOOL
VAR_INPUT
	i:INT;
END_VAR
currentIngredientName := arrayOfIngr[i].nameOfIngr;
currentWeight := STRING_TO_INT(arrayOfIngr[i].weightOfIngr);
//strCrntWay := arrayOfIngr[i].isDissolve;
way.setWay(arrayOfIngr[i].isDissolve);
ptToSwitch^.iWayIdx := way.getWayId();
currentTimeMixing := STRING_TO_TIME(arrayOfIngr[i].timeOfMixing);
message := arrayOfIngr[i].addMessage;
END_METHOD

METHOD PUBLIC checkPrgArr : BOOL
VAR_INPUT
END_VAR
currentProgramIdx:=0;
currentPrgSteps := 0;
iTotalWeight := 0;
IF LEN(arrayOfIngr[0].stepNum) = 0 THEN
		(* Поставить выброс ошибки в ответ на пустую или неправильную программу*)
		RETURN;		
END_IF
	
FOR iLine:=0 TO 100 DO		
	IF 	LEN(arrayOfIngr[iLine].stepNum) > 0 THEN
		currentPrgSteps := currentPrgSteps + 1;
		iTotalWeight := iTotalWeight + STRING_TO_INT(arrayOfIngr[iLine].weightOfIngr);
		(* Поставить выброс ошибки если вес превышает максимально допустимый *)
	ELSE
		RETURN;	
	END_IF
END_FOR
END_METHOD

METHOD PUBLIC clearList : BOOL
VAR_INPUT
END_VAR
FOR iCleanIdx:=0 TO iArrLength DO
	arrayOfIngr[iCleanIdx].stepNum:='';
	arrayOfIngr[iCleanIdx].nameOfIngr:='';
	arrayOfIngr[iCleanIdx].weightOfIngr:='';
	arrayOfIngr[iCleanIdx].isDissolve:='';
	arrayOfIngr[iCleanIdx].timeOfMixing:='';
	arrayOfIngr[iCleanIdx].addMessage:='';
END_FOR
 iCleanIdx:=0;
 iLine:=0;
END_METHOD

METHOD PUBLIC clearLine : BOOL
VAR_INPUT
END_VAR
IF iLine > 0 THEN
	iLine:=iLine - 1;
END_IF
arrayOfIngr[iLine].stepNum:='';
arrayOfIngr[iLine].nameOfIngr:='';
arrayOfIngr[iLine].weightOfIngr:='';
arrayOfIngr[iLine].isDissolve:='';
arrayOfIngr[iLine].timeOfMixing:='';
arrayOfIngr[iLine].addMessage:='';
END_METHOD

METHOD PUBLIC writeLine : BOOL
VAR_INPUT
END_VAR
arrayOfIngr[iLine].stepNum := CONCAT('Step ', INT_TO_STRING(iLine+1));
arrayOfIngr[iLine].nameOfIngr := currentIngredientName;
arrayOfIngr[iLine].weightOfIngr := INT_TO_STRING(currentWeight);
arrayOfIngr[iLine].isDissolve := way.getWay();
currentTimeMixing := TimeInput(inputTime);
arrayOfIngr[iLine].timeOfMixing := TIME_TO_STRING(currentTimeMixing);
arrayOfIngr[iLine].addMessage := message;

iLine := iLine + 1;	
IF iLine > iArrLength THEN
	iLine := 0;
END_IF
END_METHOD

END_FUNCTION_BLOCK

// Device/Application/Classes/Way
//Блок для работы с различными путями поступления ингредиентов в хоппер
FUNCTION_BLOCK Way
VAR_INPUT
END_VAR
VAR_OUTPUT
END_VAR
VAR
	iIdx:INT;
	wayList:ARRAY[0..10] OF STRING := ['Simple', 'Vibro', 'BigBag1', 'BigBag2', 'BigBag3', 'BigBag4','','','','',''];	
END_VAR

//возвращает имя текущего пути
METHOD getWay : STRING
VAR_INPUT
END_VAR
tmpLimitWay();
getWay := wayList[iIdx];
END_METHOD

METHOD PRIVATE tmpLimitWay : BOOL
VAR_INPUT
END_VAR
IF iIdx > 1 THEN
	iIdx := 1;
END_IF
END_METHOD

//Возвращает индекс текущего пути
METHOD PUBLIC getWayId : INT
VAR_INPUT
END_VAR
VAR
END_VAR
tmpLimitWay();
getWayId := iIdx;
END_METHOD

//устанавливает текущий активный путь
METHOD PUBLIC setWay : INT
VAR_INPUT
	strWay:STRING;
END_VAR
VAR
	i:INT;
END_VAR
IF LEN(strWay) = 0 THEN
	iIdx := 0;
	RETURN;
END_IF 
FOR i := 0 TO 10 DO
	IF strWay = wayList[i] THEN  //если нашли соответственное слово в массиве, устанавливаем текущий индекс этого слова
		setIdx(i);
		tmpLimitWay();
		RETURN;
	END_IF
END_FOR
END_METHOD

METHOD PRIVATE setIdx : BOOL
VAR_INPUT
	iIn:INT;
END_VAR
tmpLimitWay();
iIdx := iIn;
END_METHOD

END_FUNCTION_BLOCK

// Device/Application/Functions/TimeInput
//конвертирует DWORD во время в секундах
FUNCTION TimeInput : TIME
VAR_INPUT
	timeSet:DWORD;	
END_VAR
VAR		
END_VAR

TimeInput := DWORD_TO_TIME(timeSet * 1000);

END_FUNCTION

// Device/Application/Classes/Checker
//Проверка условий в программе
FUNCTION_BLOCK Checker
VAR_INPUT	
END_VAR
VAR_OUTPUT	
END_VAR
VAR
END_VAR

//индикатор наличия продукта в хоппере
METHOD isHopperEmpty : BOOL
VAR_INPUT
	iWeightInHopper:INT;
END_VAR
IF iWeightInHopper > 0 THEN
	isHopperEmpty := FALSE;
	ELSE
	isHopperEmpty := TRUE;
END_IF
END_METHOD

//индикатор выбранной программы
METHOD isPrgActive : BOOL
VAR_INPUT
END_VAR
IF LEN(arrayOfIngr[0].stepNum) = 0 THEN
	isPrgActive := FALSE;
	ELSE
	isPrgActive := TRUE;
END_IF
END_METHOD

END_FUNCTION_BLOCK

// Device/Application/Functions/NoiseFilter
//устраняет шумовые колебания сигнала
FUNCTION_BLOCK PUBLIC NoiseFilter
VAR_INPUT
	rIn:REAL;
	tmrStab:TON;
END_VAR
VAR_OUTPUT
	rOut:REAL;
END_VAR
VAR	
	uiMeasureAttempts: UINT := 50;
	rBig:REAL := 1;
	rSmall:REAL := 0.2;
	uiStabCount: UINT := 0;
	rUp:REAL ;
	rLow:REAL;
	bFluct:BOOL;
END_VAR

IF (isInEdges()) THEN
	IF (bFluct) THEN
		RETURN;
	ELSE		
		rOut := rIn;
		uiStabCount := uiStabCount + 1;
		IF uiStabCount > uiMeasureAttempts AND isInEdges()  THEN	
			setEdges(rBig);	
			bFluct := TRUE;
			RETURN;
		END_IF
		setEdges(rSmall);
	END_IF
ELSE
	uiStabCount := 0;
	bFluct := FALSE;
	setEdges(rBig);
		
	rOut := rIn;
	
END_IF

//проверка сигнала, находится ли он в диапазоне предельных значений шума
METHOD PRIVATE isInEdges : BOOL
VAR_INPUT
END_VAR
IF rIn < rUp AND rIn > rLow THEN
	isInEdges := TRUE;
	ELSE
	isInEdges :=  FALSE;
END_IF
END_METHOD

//устанавливает границы шума сигнала
METHOD setEdges
VAR_INPUT
	rKoef:REAL; //точная или грубая настройка
END_VAR
rUp := rIn + rKoef;
rLow := rIn - rKoef;
END_METHOD

//точность обработки сигнала
METHOD setAccuracy
VAR_INPUT
	rUpperEdge:REAL; //грубый замер
	rLowerEdge:REAL; //точный замер
END_VAR
rBig := rUpperEdge;
rSmall := rLowerEdge;
END_METHOD

METHOD PUBLIC refresh : BOOL
VAR_INPUT
END_VAR
bFluct := FALSE;
END_METHOD

END_FUNCTION_BLOCK

// Device/Application/Windows/Visualization
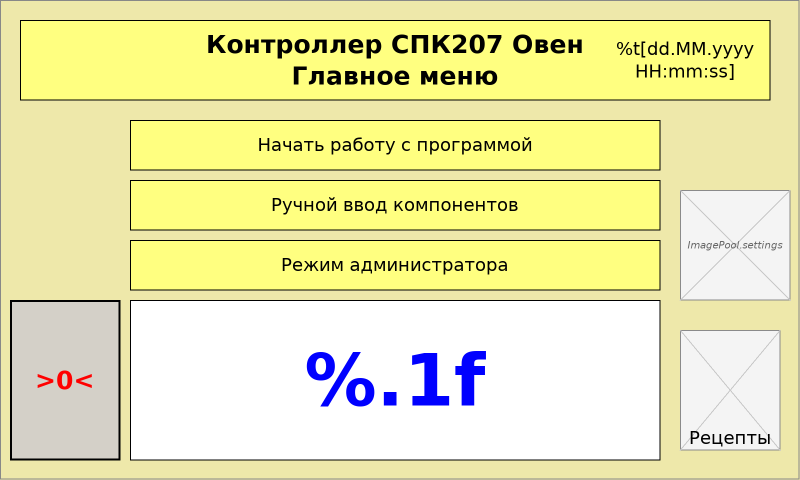
VISUALIZATION Visualization  // 800x480
    Image (680,330 100x120), "Рецепты", image: ImagePool.Iconshock-Real-Vista-Education-Laboratory
        OnMouseClick:  Assign=Settings, Type=Assignment
    RoundedRectangle (20,20 750x80), "Контроллер СПК207 Овен Главное меню", colour toggle: iInDiscrets.0
    RoundedRectangle (130,120 530x50), "Начать работу с программой"
        OnMouseClick:  Assign=AutoWork, Type=Assignment
        OnMouseClick: execute { PLC_PRG.bManMode := FALSE; PLC_PRG.actInit(); }
    RoundedRectangle (130,180 530x50), "Ручной ввод компонентов"
        OnMouseClick:  Assign=ManualInput, Type=Assignment
        OnMouseClick: execute { PLC_PRG.bManMode := TRUE; }
    RoundedRectangle (130,240 530x50), "Режим администратора"
        OnMouseClick:  Type=Login
    RoundedRectangle (130,300 530x160), "%.1f", text variable: PLC_PRG.rWeight
    RoundedRectangle (600,20 170x80), "%t[dd.MM.yyyy HH:mm:ss]"
    RoundedRectangle (10,300 110x160), ">0<"
        OnMouseClick: execute { PLC_PRG.setTara(); }
    Image (680,190 110x110), image: ImagePool.settings
        OnMouseClick:  Assign=SystemSettings, Type=Assignment
END_VISUALIZATION

// Device/Application/Windows/ManualInput
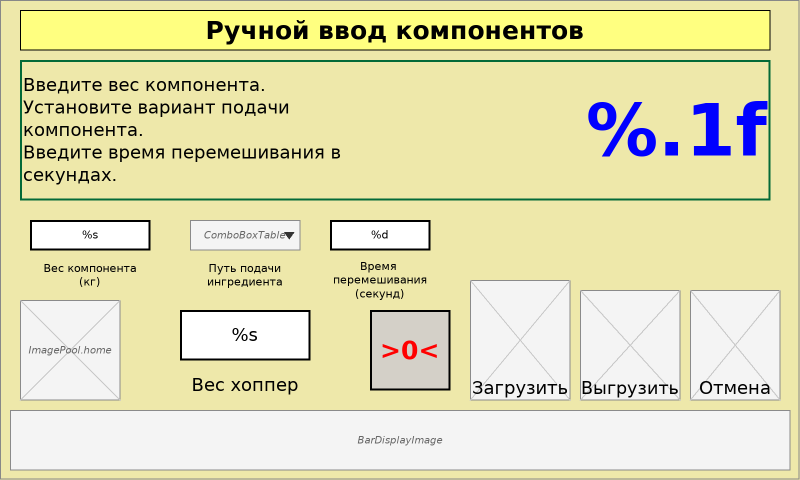
VISUALIZATION ManualInput  // 800x480
    RoundedRectangle (20,10 750x40), "Ручной ввод компонентов"
    RoundedRectangle (30,220 120x30), "%s", text variable: currentWeight, input disabled if: not PLC_PRG.checker.isHopperEmpty(PLC_PRG.x)
        OnMouseClick: write currentWeight via VisuDialogs.Numpad, min 10, max PLC_PRG.iMaxWeight
    RoundedRectangle (30,260 120x30), "Вес компонента (кг)"
    RoundedRectangle (190,260 110x30), "Путь подачи ингредиента"
    RoundedRectangle (330,220 100x30), "%d", text variable: PLC_PRG.dwInTime
        OnMouseClick: write the text variable via VisuDialogs.Numpad, min 0
    RoundedRectangle (320,260 120x40), "Время перемешивания (секунд)"
    Image (470,280 100x120), "Загрузить", image: ImagePool.download
        OnMouseClick: execute {
            PLC_PRG.bManLoadDone := FALSE;
            PLC_PRG.bRunOnce  := TRUE;
            PLC_PRG.bSwitch := TRUE;
        }
    BarDisplayImage (10,410 780x60), value: PLC_PRG.x, style: BarDisplayImage-Gray, scale format: %.0f, scale 0..1000
    RoundedRectangle (180,310 130x50), "%s", text variable: PLC_PRG.x
    Image (20,300 100x100), invisible if: not PLC_PRG.checker.isHopperEmpty(PLC_PRG.x), image: ImagePool.home
        OnMouseClick:  Assign=Visualization, Type=Assignment
        OnMouseClick: execute { PLC_PRG.bManMode := FALSE; }
    Image (580,290 100x110), "Выгрузить", image: ImagePool.upload
        OnMouseClick: execute {
            PLC_PRG.bManLoadDone := TRUE;
            PLC_PRG.bRunOnce  := TRUE;
            PLC_PRG.bSwitch := TRUE;
        }
    RoundedRectangle (180,370 130x30), "Вес хоппер"
    Image (690,290 90x110), "Отмена", image: ImagePool.cancel
        OnMouseClick: execute {
            PLC_PRG.x:=0;
            currentWeight:=0;
            PLC_PRG.dwInTime:=0;
            PLC_PRG.switch.allOff();
        }
    RoundedRectangle (20,60 750x140), "Введите вес компонента. Установите вариант подачи компонента. Введите время перемешивания в секундах."
    ComboBoxTable (190,220 110x30), variable: PLC_PRG.list.way.iIdx, input disabled if: not PLC_PRG.checker.isHopperEmpty(PLC_PRG.x), data array: PLC_PRG.list.way.wayList
        p3854506369: PLC_PRG.list.way.wayList[INDEX]
    RoundedRectangle (380,60 390x140), "%.1f", text variable: PLC_PRG.rWeight
    RoundedRectangle (370,310 80x80), ">0<"
        OnMouseClick: execute { PLC_PRG.setTara(); }
END_VISUALIZATION

// Device/Application/Windows/Settings
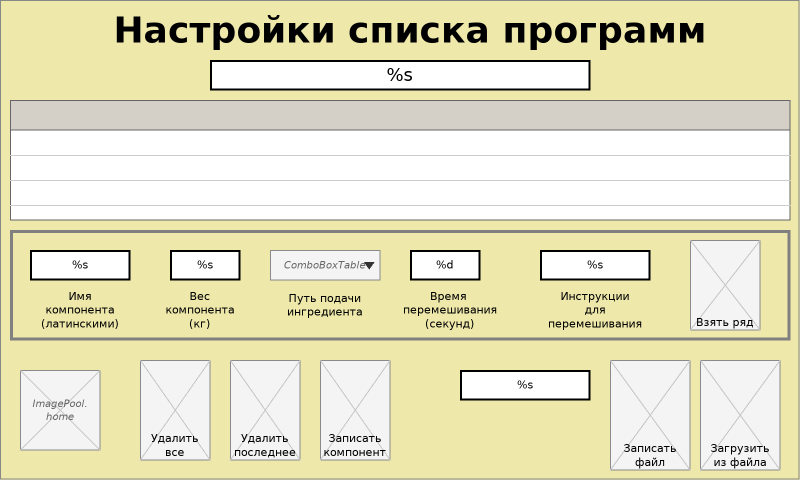
VISUALIZATION Settings  // 800x480
    Rectangle (70,10 680x40), "Настройки списка программ"
    Image (20,370 80x80), image: ImagePool.home
        OnMouseClick:  Assign=Visualization, Type=Assignment
    Rectangle (10,230 780x110)
    RoundedRectangle (170,250 70x30), "%s", text variable: currentWeight
        OnMouseClick: write currentWeight via VisuDialogs.Numpad, min 10, max PLC_PRG.iMaxWeight
    RoundedRectangle (160,280 80x60), "Вес компонента (кг)"
    RoundedRectangle (410,250 70x30), "%d", text variable: inputTime
        OnMouseClick: write the text variable via VisuDialogs.Numpad, min 0
    RoundedRectangle (390,290 120x40), "Время перемешивания (секунд)"
    RoundedRectangle (30,250 100x30), "%s", text variable: currentIngredientName
        OnMouseClick: write the text variable via Default
    RoundedRectangle (30,280 100x60), "Имя компонента (латинскими)"
    RoundedRectangle (540,250 110x30), "%s", text variable: message
        OnMouseClick: write the text variable via Default, min 1, max 30
    RoundedRectangle (530,290 130x40), "Инструкции для перемешивания"
    Image (610,360 80x110), "Записать файл", image: ImagePool.Drives-Downloads-icon
        OnMouseClick:  ExecuteCommand=ExecuteCommand=[Command=CreateRecipe, Value='Receipt', Value2=currentPrgName, Command=SaveRecipeAs, Value='Receipt', Value2=currentPrgName]
    Image (700,360 80x110), "Загрузить из файла", image: ImagePool.App-desktop-enhancements-icon
        OnMouseClick:  ExecuteCommand=ExecuteCommand=[Command=LoadRecipeFrom, Value='Receipt']
    RoundedRectangle (210,60 380x30), "%s", text variable: currentPrgName
    Image (140,360 70x100), "Удалить все", image: ImagePool.cancel
        OnMouseClick:  ExecuteCommand=ExecuteCommand=[Command=CreateRecipe, Value='Receipt', Value2='']
        OnMouseClick: execute { PLC_PRG.list.clearList(); }
    Image (230,360 70x100), "Удалить последнее", image: ImagePool.remove
        OnMouseClick: execute { PLC_PRG.list.clearLine(); }
    Image (320,360 70x100), "Записать компонент", image: ImagePool.add
        OnMouseClick: execute { PLC_PRG.list.writeLine(); }
    RoundedRectangle (460,370 130x30), "%s", text variable: currentPrgName
        OnMouseClick: write the text variable via Default, min 1, max 30
    Image (690,240 70x90), "Взять ряд", image: ImagePool.download
        OnMouseClick: execute { PLC_PRG.list.getLineFromPrgArr(PLC_PRG.list.iLine); }
    RoundedRectangle (270,290 110x30), "Путь подачи ингредиента"
    ComboBoxTable (270,250 110x30), variable: PLC_PRG.list.way.iIdx, data array: PLC_PRG.list.way.wayList
        p3854506369: PLC_PRG.list.way.wayList[INDEX]
    Table (10,100 780x120), data array: arrayOfIngr
        p3854506369: arrayOfIngr[INDEX].stepNum
        p1892666644: arrayOfIngr[INDEX].nameOfIngr
        p338671338: arrayOfIngr[INDEX].weightOfIngr
        p2170511999: arrayOfIngr[INDEX].isDissolve
        p3723444502: arrayOfIngr[INDEX].timeOfMixing
        p1218418051: arrayOfIngr[INDEX].addMessage
        p2232123230: № шага
        p511219082: Компонент
        p1755163831: Вес
        p4092479075: Путь
        p2237128397: Время
        p505689113: Инструкции
        p1137915858: PLC_PRG.list.iLine
END_VISUALIZATION

// Device/Application/Windows/AutoWork
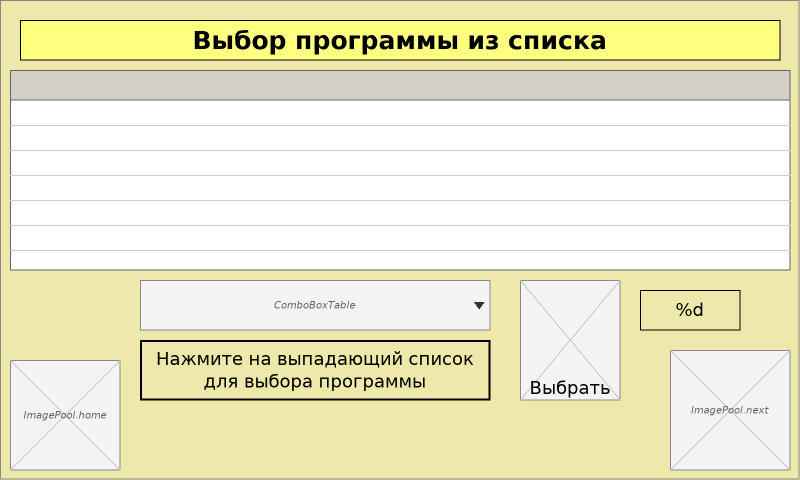
VISUALIZATION AutoWork  // 800x480
    RoundedRectangle (20,20 760x40), "Выбор программы из списка"
    Image (10,360 110x110), image: ImagePool.home
        OnMouseClick:  Assign=Visualization, Type=Assignment
    Image (520,280 100x120), "Выбрать", image: ImagePool.ok
        OnMouseClick:  ExecuteCommand=ExecuteCommand=[Command=WriteRecipe, Value='Receipt', Value2=ListOfPrgNames[PLC_PRG.list.iLinePrgList]]
        OnMouseClick: execute { PLC_PRG.list.checkPrgArr(); }
    Image (670,350 120x120), invisible if: NOT PLC_PRG.checker.isPrgActive(), image: ImagePool.next
        OnMouseClick:  Assign=LoadProcessWindow, Type=Assignment
        OnMouseClick: execute {
            PLC_PRG.bManMode := FALSE;
            currentProgramIdx:=0;
            PLC_PRG.list.getLineFromPrgArr(currentProgramIdx);
        }
    RoundedRectangle (140,340 350x60), "Нажмите на выпадающий список для выбора программы"
    ComboBoxTable (140,280 350x50), variable: PLC_PRG.list.iLinePrgList, data array: ListOfPrgNames
        p3854506369: ListOfPrgNames[INDEX]
    Rectangle (640,290 100x40), "%d", text variable: PLC_PRG.list.iTotalWeight
    Table (10,70 780x200), data array: arrayOfIngr
        p3854506369: arrayOfIngr[INDEX].stepNum
        p1892666644: arrayOfIngr[INDEX].nameOfIngr
        p338671338: arrayOfIngr[INDEX].weightOfIngr
        p2170511999: arrayOfIngr[INDEX].isDissolve
        p3723444502: arrayOfIngr[INDEX].timeOfMixing
        p1218418051: arrayOfIngr[INDEX].addMessage
        p2232123230: № шага
        p511219082: Компонент
        p1755163831: Вес
        p4092479075: Путь
        p2237128397: Время
        p505689113: Инструкции
END_VISUALIZATION

// Device/Application/Windows/LoadProcessWindow
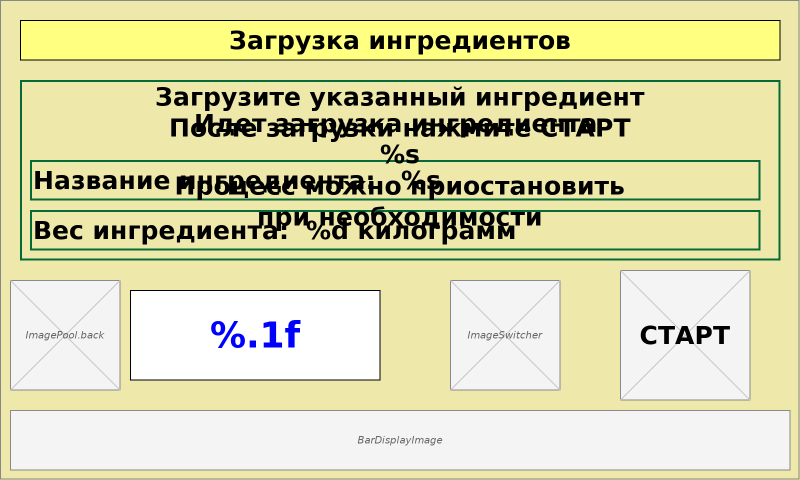
VISUALIZATION LoadProcessWindow  // 800x480
    RoundedRectangle (20,20 760x40), "Загрузка ингредиентов"
    Image (10,280 110x110), invisible if: not PLC_PRG.checker.isHopperEmpty(PLC_PRG.x), image: ImagePool.back
        OnMouseClick:  Assign=AutoWork, Type=Assignment
    BarDisplayImage (10,410 780x60), value: PLC_PRG.x, style: BarDisplayImage-Gray, scale format: %.0f, scale 0..1000
    RoundedRectangle (20,80 760x180), "Загрузите указанный ингредиент После загрузки нажмите СТАРТ", invisible if: not PLC_PRG.bMsgVisible
    RoundedRectangle (30,160 730x40), "Название ингредиента: %s", text variable: currentIngredientName, invisible if: not PLC_PRG.bMsgVisible
    RoundedRectangle (30,210 730x40), "Вес ингредиента: %d килограмм", text variable: currentWeight, invisible if: not PLC_PRG.bMsgVisible
    RoundedRectangle (20,80 760x180), "Идет загрузка ингредиента %s Процесс можно приостановить при необходимости", text variable: currentIngredientName, invisible if: PLC_PRG.bMsgVisible
    RoundedRectangle (130,290 250x90), "%.1f", text variable: PLC_PRG.rWeight
    ImageSwitcher (450,280 110x110), variable: PLC_PRG.bPause, background image: ImagePool.startAgain, image: ImagePool.pause, behaviour: TOGGLE
    Image (620,270 130x130), "СТАРТ", invisible if: not PLC_PRG.bMsgVisible, image: ImagePool.start-button-305427_960_720
        OnMouseClick:  ToggleVariable=PLC_PRG.bSwitch
END_VISUALIZATION

// Device/Application/Windows/LoadingFinished
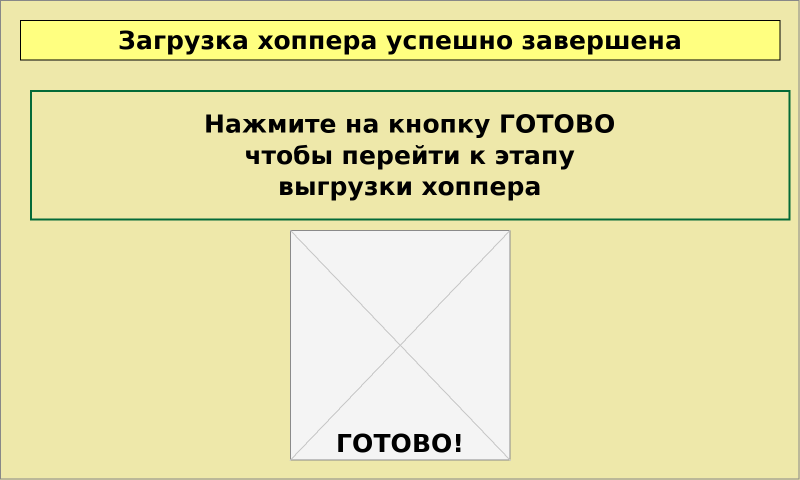
VISUALIZATION LoadingFinished  // 800x480
    RoundedRectangle (20,20 760x40), "Загрузка хоппера успешно завершена"
    Image (290,230 220x230), "ГОТОВО!", image: ImagePool.ok
        OnMouseClick:  Assign=UnloadProcessWindow, Type=Assignment
        OnMouseClick: execute { PLC_PRG.bLoadDone := TRUE; }
    RoundedRectangle (30,90 760x130), "Нажмите на кнопку ГОТОВО чтобы перейти к этапу выгрузки хоппера"
END_VISUALIZATION

// Device/Application/Windows/UnloadProcessWindow
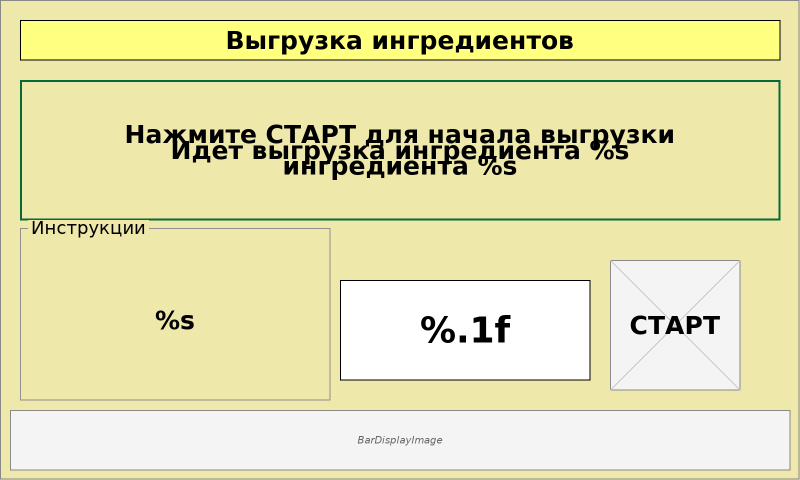
VISUALIZATION UnloadProcessWindow  // 800x480
    RoundedRectangle (20,20 760x40), "Выгрузка ингредиентов"
    BarDisplayImage (10,410 780x60), value: PLC_PRG.x, style: BarDisplayImage-Gray, scale format: %.0f, scale 0..1000
    RoundedRectangle (20,80 760x140), "Идет выгрузка ингредиента %s", text variable: currentIngredientName, invisible if: PLC_PRG.bMsgVisible
    RoundedRectangle (20,80 760x140), "Нажмите СТАРТ для начала выгрузки ингредиента %s", text variable: currentIngredientName, invisible if: not PLC_PRG.bMsgVisible
    Image (610,260 130x130), "СТАРТ", invisible if: not PLC_PRG.bMsgVisible, image: ImagePool.start-button-305427_960_720
        OnMouseClick:  ToggleVariable=PLC_PRG.bSwitch
    RoundedRectangle (20,240 310x160), "%s", text variable: message, invisible if: not PLC_PRG.bMsgVisible
    GroupBox (20,220 310x180), "Инструкции"
    RoundedRectangle (340,280 250x100), "%.1f", text variable: PLC_PRG.rWeight
END_VISUALIZATION

// Device/Application/Windows/RepeatOrNewPRG
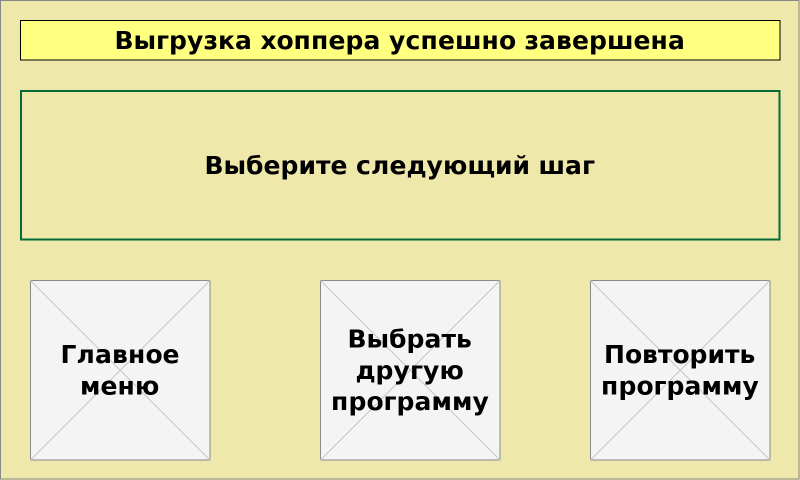
VISUALIZATION RepeatOrNewPRG  // 800x480
    RoundedRectangle (20,20 760x40), "Выгрузка хоппера успешно завершена"
    Image (320,280 180x180), "Выбрать другую программу", image: ImagePool.add
        OnMouseClick:  Assign=AutoWork, Type=Assignment
        OnMouseClick: execute { PLC_PRG.bLoadDone:=false; }
    RoundedRectangle (20,90 760x150), "Выберите следующий шаг"
    Image (30,280 180x180), "Главное меню", image: ImagePool.home
        OnMouseClick:  Assign=Visualization, Type=Assignment
    Image (590,280 180x180), "Повторить программу", image: ImagePool.repeat
        OnMouseClick:  Assign=LoadProcessWindow, Type=Assignment
        OnMouseClick: execute {
            PLC_PRG.bLoadDone:=FALSE;
            currentProgramIdx:=0;
            PLC_PRG.list.getLineFromPrgArr(currentProgramIdx);
        }
END_VISUALIZATION

// Device/Application/Windows/TimeCounter
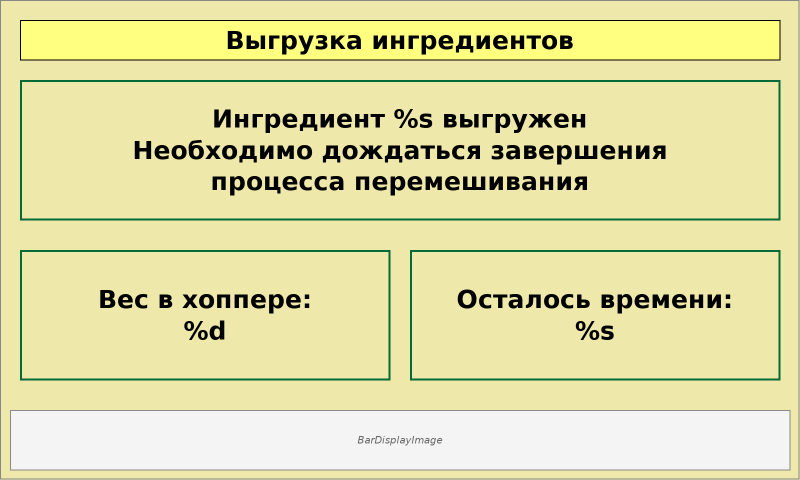
VISUALIZATION TimeCounter  // 800x480
    BarDisplayImage (10,410 780x60), value: PLC_PRG.x, style: BarDisplayImage-Gray, scale format: %.0f, scale 0..1000
    RoundedRectangle (20,80 760x140), "Ингредиент %s выгружен Необходимо дождаться завершения процесса перемешивания", text variable: currentIngredientName, invisible if: not PLC_PRG.bMsgVisible
    RoundedRectangle (20,20 760x40), "Выгрузка ингредиентов"
    RoundedRectangle (410,250 370x130), "Осталось времени: %s", text variable: PLC_PRG.strTimer, invisible if: not PLC_PRG.bMsgVisible
    RoundedRectangle (20,250 370x130), "Вес в хоппере: %d", text variable: PLC_PRG.x, invisible if: not PLC_PRG.bMsgVisible
END_VISUALIZATION

// Device/Application/Windows/Dialogs/DialogLoad
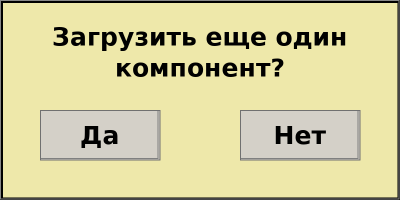
VISUALIZATION DialogLoad  // 400x200
    RoundedRectangle (0,0 400x200)
    Rectangle (0,20 400x70), "Загрузить еще один компонент?"
    Button (40,110 120x50), "Да"
        OnMouseClick:  Dialog=DialogLoad, Result=OK, NumpadKeypadSet=True
    Button (240,110 120x50), "Нет"
        OnMouseClick:  Dialog=DialogLoad, Result=OK, NumpadKeypadSet=True
END_VISUALIZATION

// Device/Application/Windows/TmpUnused
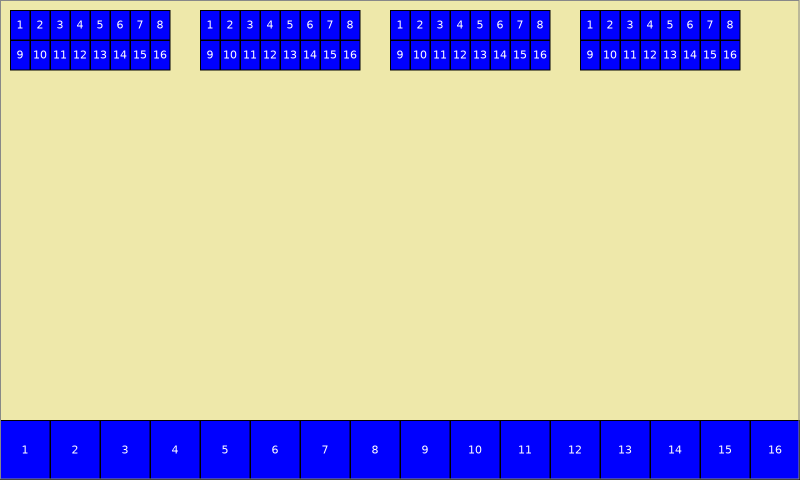
VISUALIZATION TmpUnused  // 800x480
    Rectangle (10,10 20x30), "1", colour toggle: PLC_PRG.switch.iOut.0
    Rectangle (30,10 20x30), "2", colour toggle: PLC_PRG.switch.iOut.1
    Rectangle (50,10 20x30), "3", colour toggle: PLC_PRG.switch.iOut.2
    Rectangle (70,10 20x30), "4", colour toggle: PLC_PRG.switch.iOut.3
    Rectangle (90,10 20x30), "5", colour toggle: PLC_PRG.switch.iOut.4
    Rectangle (110,10 20x30), "6", colour toggle: PLC_PRG.switch.iOut.5
    Rectangle (130,10 20x30), "7", colour toggle: PLC_PRG.switch.iOut.6
    Rectangle (150,10 20x30), "8", colour toggle: PLC_PRG.switch.iOut.7
    Rectangle (10,40 20x30), "9", colour toggle: PLC_PRG.switch.iOut.8
    Rectangle (30,40 20x30), "10", colour toggle: PLC_PRG.switch.iOut.9
    Rectangle (50,40 20x30), "11", colour toggle: PLC_PRG.switch.iOut.10
    Rectangle (70,40 20x30), "12", colour toggle: PLC_PRG.switch.iOut.11
    Rectangle (90,40 20x30), "13", colour toggle: PLC_PRG.switch.iOut.12
    Rectangle (110,40 20x30), "14", colour toggle: PLC_PRG.switch.iOut.13
    Rectangle (130,40 20x30), "15", colour toggle: PLC_PRG.switch.iOut.14
    Rectangle (150,40 20x30), "16", colour toggle: PLC_PRG.switch.iOut.15
    Rectangle (200,10 20x30), "1", colour toggle: PLC_PRG.switch.iOut.0
    Rectangle (220,10 20x30), "2", colour toggle: PLC_PRG.switch.iOut.1
    Rectangle (240,10 20x30), "3", colour toggle: PLC_PRG.switch.iOut.2
    Rectangle (260,10 20x30), "4", colour toggle: PLC_PRG.switch.iOut.3
    Rectangle (280,10 20x30), "5", colour toggle: PLC_PRG.switch.iOut.4
    Rectangle (300,10 20x30), "6", colour toggle: PLC_PRG.switch.iOut.5
    Rectangle (320,10 20x30), "7", colour toggle: PLC_PRG.switch.iOut.6
    Rectangle (340,10 20x30), "8", colour toggle: PLC_PRG.switch.iOut.7
    Rectangle (200,40 20x30), "9", colour toggle: PLC_PRG.switch.iOut.8
    Rectangle (220,40 20x30), "10", colour toggle: PLC_PRG.switch.iOut.9
    Rectangle (240,40 20x30), "11", colour toggle: PLC_PRG.switch.iOut.10
    Rectangle (260,40 20x30), "12", colour toggle: PLC_PRG.switch.iOut.11
    Rectangle (280,40 20x30), "13", colour toggle: PLC_PRG.switch.iOut.12
    Rectangle (300,40 20x30), "14", colour toggle: PLC_PRG.switch.iOut.13
    Rectangle (320,40 20x30), "15", colour toggle: PLC_PRG.switch.iOut.14
    Rectangle (340,40 20x30), "16", colour toggle: PLC_PRG.switch.iOut.15
    Rectangle (390,10 20x30), "1", colour toggle: PLC_PRG.switch.iOut.0
    Rectangle (410,10 20x30), "2", colour toggle: PLC_PRG.switch.iOut.1
    Rectangle (430,10 20x30), "3", colour toggle: PLC_PRG.switch.iOut.2
    Rectangle (450,10 20x30), "4", colour toggle: PLC_PRG.switch.iOut.3
    Rectangle (470,10 20x30), "5", colour toggle: PLC_PRG.switch.iOut.4
    Rectangle (490,10 20x30), "6", colour toggle: PLC_PRG.switch.iOut.5
    Rectangle (510,10 20x30), "7", colour toggle: PLC_PRG.switch.iOut.6
    Rectangle (530,10 20x30), "8", colour toggle: PLC_PRG.switch.iOut.7
    Rectangle (390,40 20x30), "9", colour toggle: PLC_PRG.switch.iOut.8
    Rectangle (410,40 20x30), "10", colour toggle: PLC_PRG.switch.iOut.9
    Rectangle (430,40 20x30), "11", colour toggle: PLC_PRG.switch.iOut.10
    Rectangle (450,40 20x30), "12", colour toggle: PLC_PRG.switch.iOut.11
    Rectangle (470,40 20x30), "13", colour toggle: PLC_PRG.switch.iOut.12
    Rectangle (490,40 20x30), "14", colour toggle: PLC_PRG.switch.iOut.13
    Rectangle (510,40 20x30), "15", colour toggle: PLC_PRG.switch.iOut.14
    Rectangle (530,40 20x30), "16", colour toggle: PLC_PRG.switch.iOut.15
    Rectangle (580,10 20x30), "1", colour toggle: PLC_PRG.switch.iOut.0
    Rectangle (600,10 20x30), "2", colour toggle: PLC_PRG.switch.iOut.1
    Rectangle (620,10 20x30), "3", colour toggle: PLC_PRG.switch.iOut.2
    Rectangle (640,10 20x30), "4", colour toggle: PLC_PRG.switch.iOut.3
    Rectangle (660,10 20x30), "5", colour toggle: PLC_PRG.switch.iOut.4
    Rectangle (680,10 20x30), "6", colour toggle: PLC_PRG.switch.iOut.5
    Rectangle (700,10 20x30), "7", colour toggle: PLC_PRG.switch.iOut.6
    Rectangle (720,10 20x30), "8", colour toggle: PLC_PRG.switch.iOut.7
    Rectangle (580,40 20x30), "9", colour toggle: PLC_PRG.switch.iOut.8
    Rectangle (600,40 20x30), "10", colour toggle: PLC_PRG.switch.iOut.9
    Rectangle (620,40 20x30), "11", colour toggle: PLC_PRG.switch.iOut.10
    Rectangle (640,40 20x30), "12", colour toggle: PLC_PRG.switch.iOut.11
    Rectangle (660,40 20x30), "13", colour toggle: PLC_PRG.switch.iOut.12
    Rectangle (680,40 20x30), "14", colour toggle: PLC_PRG.switch.iOut.13
    Rectangle (700,40 20x30), "15", colour toggle: PLC_PRG.switch.iOut.14
    Rectangle (720,40 20x30), "16", colour toggle: PLC_PRG.switch.iOut.15
    Rectangle (0,420 50x60), "1", colour toggle: PLC_PRG.switch.iOut.0
        OnMouseClick:  ToggleVariable=PLC_PRG.switch.iOut.0
    Rectangle (50,420 50x60), "2", colour toggle: PLC_PRG.switch.iOut.1
        OnMouseClick:  ToggleVariable=PLC_PRG.switch.iOut.1
    Rectangle (100,420 50x60), "3", colour toggle: PLC_PRG.switch.iOut.2
        OnMouseClick:  ToggleVariable=PLC_PRG.switch.iOut.2
    Rectangle (150,420 50x60), "4", colour toggle: PLC_PRG.switch.iOut.3
        OnMouseClick:  ToggleVariable=PLC_PRG.switch.iOut.3
    Rectangle (200,420 50x60), "5", colour toggle: PLC_PRG.switch.iOut.4
        OnMouseClick:  ToggleVariable=PLC_PRG.switch.iOut.4
    Rectangle (250,420 50x60), "6", colour toggle: PLC_PRG.switch.iOut.5
        OnMouseClick:  ToggleVariable=PLC_PRG.switch.iOut.5
    Rectangle (300,420 50x60), "7", colour toggle: PLC_PRG.switch.iOut.6
        OnMouseClick:  ToggleVariable=PLC_PRG.switch.iOut.6
    Rectangle (350,420 50x60), "8", colour toggle: PLC_PRG.switch.iOut.7
        OnMouseClick:  ToggleVariable=PLC_PRG.switch.iOut.7
    Rectangle (400,420 50x60), "9", colour toggle: PLC_PRG.switch.iOut.8
        OnMouseClick:  ToggleVariable=PLC_PRG.switch.iOut.8
    Rectangle (450,420 50x60), "10", colour toggle: PLC_PRG.switch.iOut.9
        OnMouseClick:  ToggleVariable=PLC_PRG.switch.iOut.9
    Rectangle (500,420 50x60), "11", colour toggle: PLC_PRG.switch.iOut.10
        OnMouseClick:  ToggleVariable=PLC_PRG.switch.iOut.10
    Rectangle (550,420 50x60), "12", colour toggle: PLC_PRG.switch.iOut.11
        OnMouseClick:  ToggleVariable=PLC_PRG.switch.iOut.11
    Rectangle (600,420 50x60), "13", colour toggle: PLC_PRG.switch.iOut.12
        OnMouseClick:  ToggleVariable=PLC_PRG.switch.iOut.12
    Rectangle (650,420 50x60), "14", colour toggle: PLC_PRG.switch.iOut.13
        OnMouseClick:  ToggleVariable=PLC_PRG.switch.iOut.13
    Rectangle (700,420 50x60), "15", colour toggle: PLC_PRG.switch.iOut.14
        OnMouseClick:  ToggleVariable=PLC_PRG.switch.iOut.14
    Rectangle (750,420 50x60), "16", colour toggle: PLC_PRG.switch.iOut.15
        OnMouseClick:  ToggleVariable=PLC_PRG.switch.iOut.15
END_VISUALIZATION

// Device/Application/Windows/SystemSettings
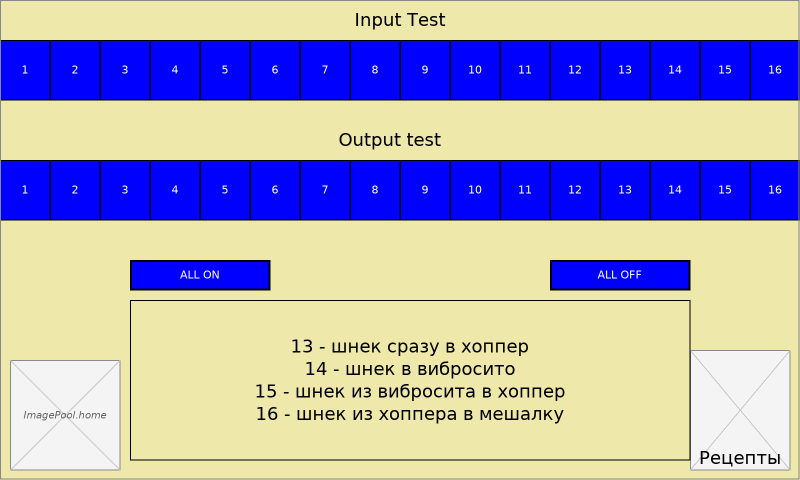
VISUALIZATION SystemSettings  // 800x480
    Rectangle (0,40 50x60), "1", colour toggle: PLC_PRG.switch.iIn.0
    Rectangle (50,40 50x60), "2", colour toggle: PLC_PRG.switch.iIn.1
    Rectangle (100,40 50x60), "3", colour toggle: PLC_PRG.switch.iIn.2
    Rectangle (150,40 50x60), "4", colour toggle: PLC_PRG.switch.iIn.3
    Rectangle (200,40 50x60), "5", colour toggle: PLC_PRG.switch.iIn.4
    Rectangle (250,40 50x60), "6", colour toggle: PLC_PRG.switch.iIn.5
    Rectangle (300,40 50x60), "7", colour toggle: PLC_PRG.switch.iIn.6
    Rectangle (350,40 50x60), "8", colour toggle: PLC_PRG.switch.iIn.7
    Rectangle (400,40 50x60), "9", colour toggle: PLC_PRG.switch.iIn.8
    Rectangle (450,40 50x60), "10", colour toggle: PLC_PRG.switch.iIn.9
    Rectangle (500,40 50x60), "11", colour toggle: PLC_PRG.switch.iIn.10
    Rectangle (550,40 50x60), "12", colour toggle: PLC_PRG.switch.iIn.11
    Rectangle (600,40 50x60), "13", colour toggle: PLC_PRG.switch.iIn.12
    Rectangle (650,40 50x60), "14", colour toggle: PLC_PRG.switch.iIn.13
    Rectangle (700,40 50x60), "15", colour toggle: PLC_PRG.switch.iIn.14
    Rectangle (750,40 50x60), "16", colour toggle: PLC_PRG.switch.iIn.15
    Image (10,360 110x110), image: ImagePool.home
        OnMouseClick:  Assign=Visualization, Type=Assignment
    Image (690,350 100x120), "Рецепты", image: ImagePool.Iconshock-Real-Vista-Education-Laboratory
        OnMouseClick:  Assign=Settings, Type=Assignment
    Rectangle (0,160 50x60), "1", colour toggle: PLC_PRG.switch.iOut.0
        OnMouseClick:  ToggleVariable=PLC_PRG.switch.iOut.0
    Rectangle (50,160 50x60), "2", colour toggle: PLC_PRG.switch.iOut.1
        OnMouseClick:  ToggleVariable=PLC_PRG.switch.iOut.1
    Rectangle (100,160 50x60), "3", colour toggle: PLC_PRG.switch.iOut.2
        OnMouseClick:  ToggleVariable=PLC_PRG.switch.iOut.2
    Rectangle (150,160 50x60), "4", colour toggle: PLC_PRG.switch.iOut.3
        OnMouseClick:  ToggleVariable=PLC_PRG.switch.iOut.3
    Rectangle (200,160 50x60), "5", colour toggle: PLC_PRG.switch.iOut.4
        OnMouseClick:  ToggleVariable=PLC_PRG.switch.iOut.4
    Rectangle (250,160 50x60), "6", colour toggle: PLC_PRG.switch.iOut.5
        OnMouseClick:  ToggleVariable=PLC_PRG.switch.iOut.5
    Rectangle (300,160 50x60), "7", colour toggle: PLC_PRG.switch.iOut.6
        OnMouseClick:  ToggleVariable=PLC_PRG.switch.iOut.6
    Rectangle (350,160 50x60), "8", colour toggle: PLC_PRG.switch.iOut.7
        OnMouseClick:  ToggleVariable=PLC_PRG.switch.iOut.7
    Rectangle (400,160 50x60), "9", colour toggle: PLC_PRG.switch.iOut.8
        OnMouseClick:  ToggleVariable=PLC_PRG.switch.iOut.8
    Rectangle (450,160 50x60), "10", colour toggle: PLC_PRG.switch.iOut.9
        OnMouseClick:  ToggleVariable=PLC_PRG.switch.iOut.9
    Rectangle (500,160 50x60), "11", colour toggle: PLC_PRG.switch.iOut.10
        OnMouseClick:  ToggleVariable=PLC_PRG.switch.iOut.10
    Rectangle (550,160 50x60), "12", colour toggle: PLC_PRG.switch.iOut.11
        OnMouseClick:  ToggleVariable=PLC_PRG.switch.iOut.11
    Rectangle (600,160 50x60), "13", colour toggle: PLC_PRG.switch.iOut.12
        OnMouseClick:  ToggleVariable=PLC_PRG.switch.iOut.12
    Rectangle (650,160 50x60), "14", colour toggle: PLC_PRG.switch.iOut.13
        OnMouseClick:  ToggleVariable=PLC_PRG.switch.iOut.13
    Rectangle (700,160 50x60), "15", colour toggle: PLC_PRG.switch.iOut.14
        OnMouseClick:  ToggleVariable=PLC_PRG.switch.iOut.14
    Rectangle (750,160 50x60), "16", colour toggle: PLC_PRG.switch.iOut.15
        OnMouseClick:  ToggleVariable=PLC_PRG.switch.iOut.15
    Rectangle (160,0 480x40), "Input Test"
    Rectangle (150,120 480x40), "Output test"
    RoundedRectangle (130,260 140x30), "ALL ON"
        OnMouseClick: execute { PLC_PRG.switch.iOut := 65535; }
    RoundedRectangle (550,260 140x30), "ALL OFF"
        OnMouseClick: execute { PLC_PRG.switch.iOut := 0; }
    RoundedRectangle (130,300 560x160), "13 - шнек сразу в хоппер 14 - шнек в вибросито 15 - шнек из вибросита в хоппер 16 - шнек из хоппера в мешалку"
END_VISUALIZATION

// Device/Application/Windows/Dialogs/Alarm
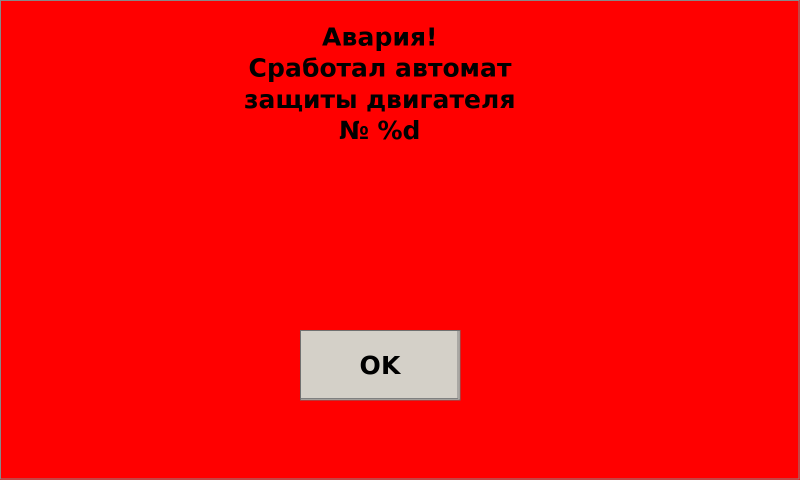
VISUALIZATION Alarm  // 800x480
    Rectangle (180,20 400x200), "Авария! Сработал автомат защиты двигателя № %d", text variable: PLC_PRG.iErrEngineNum
    Button (300,330 160x70), "OK"
        OnMouseClick:  Assign=Visualization, Type=Previous
        OnMouseClick: execute {
            IF PLC_PRG.bSwitch THEN
            	PLC_PRG.switch.set(ON);
            END_IF
        }
END_VISUALIZATION
